FUNCTION_BLOCK FB_Transport
VAR_INPUT
	bEnable : BOOL;
	bExecute : BOOL;
	nStation : INT;
	
	bSens1 : BOOL;
	bSens2 : BOOL;
	bSens3 : BOOL;
	bSens4 : BOOL;
END_VAR
VAR_OUTPUT
	eState : eBetriebszustand;
	
	bStopper1 : BOOL;
	bStopper2 : BOOL;
	bStopper3 : BOOL;
END_VAR
VAR
	fbTransportE : FB_TransportE;
	fbTransportLogik : FB_TransportLogik;
	fbTransportBand : FB_Forderband;
	fbTransportA : FB_TransportA;
END_VAR
VAR_IN_OUT
    ax : AXIS_REF;
END_VAR

fbTransportE(
	bSens1:= bSens1, 
	bSens2:= bSens2, 
	bSens3:= bSens3, 
	bSens4:= bSens4, 
	bStation1=> , 
	bStation2=> , 
	bStation3=> , 
	bStation4=> );
	
fbTransportLogik(
	eStateE:= fbTransportBand.eState, 
	bEnable:= bEnable, 
	bExecute:= bExecute, 
	nStation:= nStation, 
	bStation1:= fbTransportE.bStation1, 
	bStation2:= fbTransportE.bStation2, 
	bStation3:= fbTransportE.bStation3, 
	bStation4:= fbTransportE.bStation4, 
	eStateA=> eState, 
	bEnableA=> , 
	bExecuteA=> , 
	bHaltA=> , 
	bStop1=> , 
	bStop2=> , 
	bStop3=> );
	
fbTransportBand(
	bEnable:= fbTransportLogik.bEnableA, 
	bExecute:= fbTransportLogik.bExecuteA, 
	bHalt:= fbTransportLogik.bHaltA, 
	eState=> , 
	ax:= ax);
	
fbTransportA(
	bStop1:= fbTransportLogik.bStop1, 
	bStop2:= fbTransportLogik.bStop2, 
	bStop3:= fbTransportLogik.bStop3, 
	bStopper1=> bStopper1, 
	bStopper2=> bStopper2, 
	bStopper3=> bStopper3);

END_FUNCTION_BLOCK

(* stored: Version 1.1.0.1, ProductVersion 3.1.4024.15
   POU FB_Transport: Id {d1b3ac44-c26b-481c-9208-f5c59357332a}, SpecialFunc None *)
